// TIA Portal project "Programa" (V19)

(* hardware
DEVICE "S7-1200 station_1"  S7-1200 Station
   slot 0: "Rack_0"  S7-1200 Rack  Rack  V1.0
   slot 1: "PLC_1"  CPU 1212C DC/DC/DC  6ES7 212-1AE40-0XB0  V4.6
DEVICE "HMI_1"  KTP400 Basic PN
   slot 0: "HMI_1"  KTP400 Basic PN  6AV2 123-2DB03-0AX0  15.1.0.0
   slot 1: "HMI_RT_1"  KTP400 Basic PN  6AV2 123-2DB03-0AX0  15.1.0.0
   slot 5: "HMI_1.IE_CP_1"  PROFINET Interface  15.0.1.0
      slot 1: "Interfaz PROFINET_1"  PROFINET Interface
         slot 1: "Port_1"  Port
*)

// ===== PLC "PLC_1"  CPU 1212C DC/DC/DC =====

VAR_GLOBAL   // PLC tag table "Default tag table"
   "Pulsador_2" AT %I0.0 : Bool;
   "Luz_2_G" AT %Q0.3 : Bool;
   "Pulsador_1" AT %I0.4 : Bool;
   "Luz_1_Y" AT %Q0.4 : Bool;
   "Paro_Emergencia" AT %I0.1 : Bool;
   "Pulsador_Stop" AT %I0.3 : Bool;
   "Pulsador_Start" AT %I0.2 : Bool;
   "Potenciometro_1" AT %IW64 : Int;
   "Potenciometro_2" AT %IW66 : Int;
   "Valor_Pot_1" AT %MD56 : Real;
   "Voltaje_1" AT %MD34 : Real;
   "Valor_Pot_2" AT %MD38 : Real;
   "Voltaje_2" AT %MD46 : Real;
   "Eje_1_Impulso" AT %Q0.0 : Bool;
   "Eje_1_Sentido" AT %Q0.1 : Bool;
   "Eje_1_HabilitarAccionamiento" AT %Q0.2 : Bool;
   "System_Byte" AT %MB1 : Byte;
   "FirstScan" AT %M1.0 : Bool;
   "DiagStatusUpdate" AT %M1.1 : Bool;
   "AlwaysTRUE" AT %M1.2 : Bool;
   "AlwaysFALSE" AT %M1.3 : Bool;
   "Clock_Byte" AT %MB0 : Byte;
   "Clock_10Hz" AT %M0.0 : Bool;
   "Clock_5Hz" AT %M0.1 : Bool;
   "Clock_2.5Hz" AT %M0.2 : Bool;
   "Clock_2Hz" AT %M0.3 : Bool;
   "Clock_1.25Hz" AT %M0.4 : Bool;
   "Clock_1Hz" AT %M0.5 : Bool;
   "Clock_0.625Hz" AT %M0.6 : Bool;
   "Clock_0.5Hz" AT %M0.7 : Bool;
   "Activación_Motor" AT %M2.0 : Bool;
   "Dirección_Motor" AT %M2.1 : Bool;
   "Set_Home" AT %M2.2 : Bool;
   "Detención_Eje" AT %M2.3 : Bool;
   "Activación_Modo_Relativo" AT %M2.4 : Bool;
   "Rotación_Motor" AT %MD10 : Real;
   "Velocidad_Motor" AT %MD14 : Real;
   "Activación_Modo_Absoluto" AT %M2.5 : Bool;
   "Tag_7" AT %MD18 : Real;
   "Tag_8" AT %MD22 : Real;
   "Activacion_Modo_Velocidad" AT %M2.6 : Bool;
   "Dir_Motor" AT %MW26 : Int;
   "Dirección_Izquierda" AT %M3.0 : Bool;
   "Dirección_Derecha" AT %M3.1 : Bool;
   "HMI_Activación" AT %M3.2 : Bool;
   "Vel_Norm" AT %MW28 : Int;
   "Set_vel_Norm" AT %MW30 : Int;
   "Luz_3_R" AT %Q0.5 : Bool;
   "Luz_Verde" AT %M3.3 : Bool;
   "Luz_Amarilla" AT %M3.4 : Bool;
   "Luz_Roja" AT %M3.5 : Bool;
   "Eje_Detenido" AT %M3.6 : Bool;
   "Eje_Trabajando" AT %M3.7 : Bool;
   "Izq_HMI" AT %M4.0 : Bool;
   "Der_HMI" AT %M4.1 : Bool;
   "Pulsos_Nor" AT %MD42 : Real;
   "Rotacion_Norm" AT %MW50 : Int;
   "Activar_Pot" AT %M4.2 : Bool;
   "Vel_pot" AT %MW52 : Int;
END_VAR

DATA_BLOCK "Eje_1"   // DB1, Motion_DB
{ S7_Optimized_Access := 'TRUE' }
AUTHOR : SIMATIC
FAMILY : BasicMC
NAME : TO_PosAx
VERSION : 8.0
// stored: InstanceOfName TO_PositioningAxis
"TO_PositioningAxis"
BEGIN
   // Axis.EnableOutput_AddressCU = %Q0.2
   // Axis.LengthUnit.LastDistance = -1
   // Axis.OnlinePtoModeCU = 16#0000_0002
   // Axis.DirectionOutputEnabledCU = TRUE
   // Axis.SelectedChannel2EnumCU = %Q0.1
   // Axis.SelectedChannel1EnumCU = %Q0.0
   // Pulse.MinDeltaDeltaFrequencyCU = 0.004
   // Pulse.MaxDeltaDeltaFrequencyCU = 1.0E+10
   // Pulse.MinDeltaFrequencyCU = 0.005
   // Pulse.MaxDeltaFrequencyCU = 9.5E+9
   // Pulse.MinFrequencyCU = 1.0
   // Pulse.MaxFrequencyCU = 100000.0
   // Pulse.OutputSourceCU = 16#0000_0000
   // Axis.SelectPTO = 0
END_DATA_BLOCK

ORGANIZATION_BLOCK "Main"   // OB1, LAD, ProgramCycle
TITLE = "Main Program Sweep (Cycle)"
{ S7_Optimized_Access := 'TRUE' }
VERSION : 0.1
   VAR_INPUT
      Initial_Call : Bool;   // Initial call of this OB
      Remanence : Bool;   // =True, if remanent data are available
   END_VAR
BEGIN

REGION Network 1
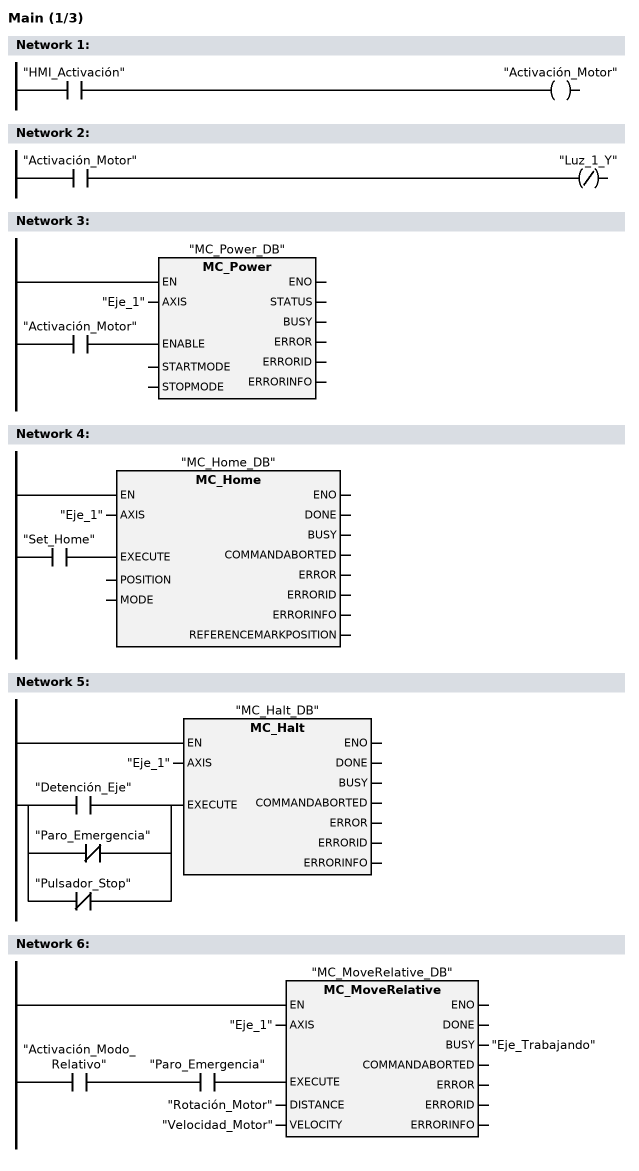
   RUNG wire#powerrail
      Contact( "HMI_Activación" )
      Coil( "Activación_Motor" )
   END_RUNG
   // the same network as SCL:
   "Activación_Motor" := "HMI_Activación";
END_REGION

REGION Network 2
   RUNG wire#powerrail
      Contact( "Activación_Motor" )
      I_Coil( "Luz_1_Y" )
   END_RUNG
   // the same network as SCL:
   "Luz_1_Y" := NOT "Activación_Motor";
END_REGION

REGION Network 3
   "MC_Power_DB"(Axis := "Eje_1", Enable := "Activación_Motor");   // MC_Power
END_REGION

REGION Network 4
   "MC_Home_DB"(Axis := "Eje_1", Execute := "Set_Home");   // MC_Home
END_REGION

REGION Network 5
   "MC_Halt_DB"(Axis := "Eje_1", Execute := "Detención_Eje" OR NOT "Paro_Emergencia" OR NOT "Pulsador_Stop");   // MC_Halt
END_REGION

REGION Network 6
   "MC_MoveRelative_DB"(Axis := "Eje_1",   // MC_MoveRelative
                        Execute := "Activación_Modo_Relativo" AND "Paro_Emergencia",
                        Distance := "Rotación_Motor",
                        Velocity := "Velocidad_Motor",
                        Busy => "Eje_Trabajando");
END_REGION

REGION Network 7
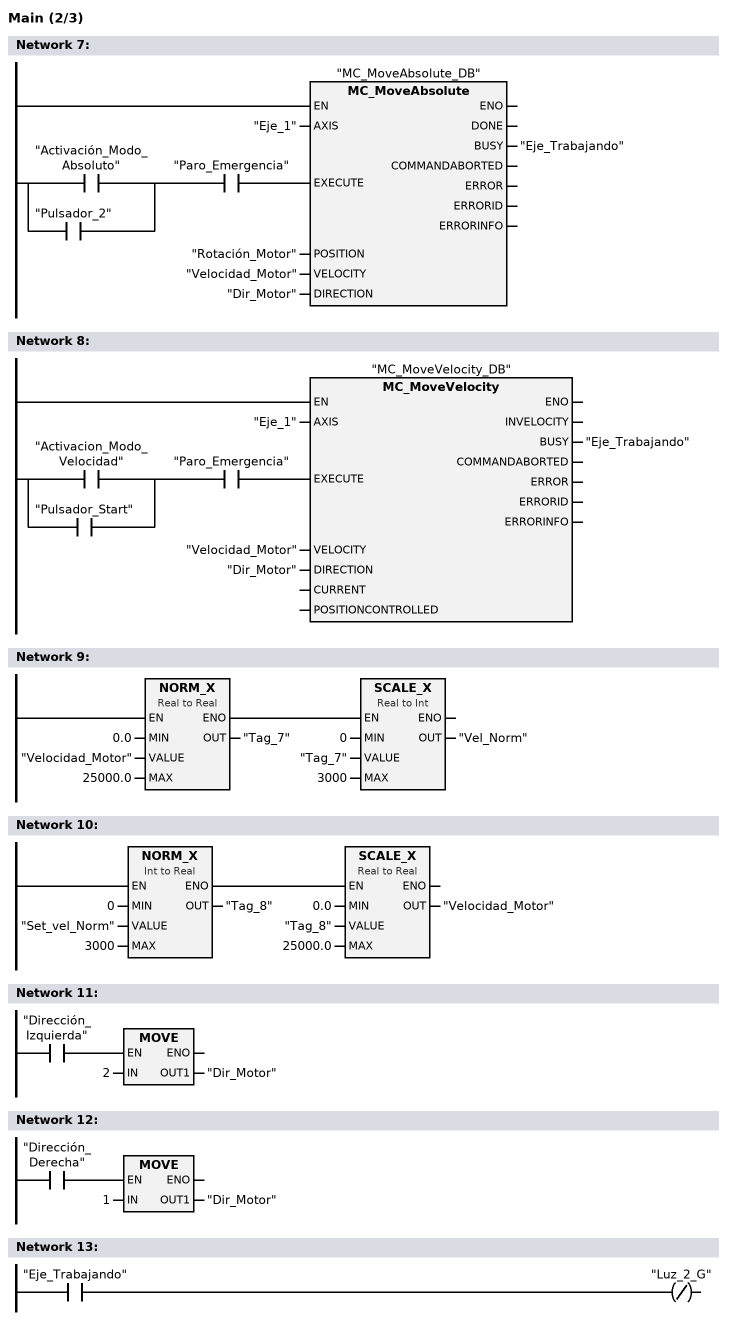
   "MC_MoveAbsolute_DB"(Axis := "Eje_1",   // MC_MoveAbsolute
                        Execute := ("Activación_Modo_Absoluto" OR "Pulsador_2") AND "Paro_Emergencia",
                        Position := "Rotación_Motor",
                        Velocity := "Velocidad_Motor",
                        Direction := "Dir_Motor",
                        Busy => "Eje_Trabajando");
END_REGION

REGION Network 8
   "MC_MoveVelocity_DB"(Axis := "Eje_1",   // MC_MoveVelocity
                        Execute := ("Activacion_Modo_Velocidad" OR "Pulsador_Start") AND "Paro_Emergencia",
                        Velocity := "Velocidad_Motor",
                        Direction := "Dir_Motor",
                        Busy => "Eje_Trabajando");
END_REGION

REGION Network 9
   RUNG wire#powerrail
      { S7_Templates := "[SrcType := Real, DestType := Real]" } Normalize(min := 0.0, value := "Velocidad_Motor", max := 25000.0, out => "Tag_7")
      { S7_Templates := "[SrcType := Real, DestType := Int]" } Scale(min := 0, value := "Tag_7", max := 3000, out => "Vel_Norm")
   END_RUNG
   // the same network as SCL:
   "Tag_7" := NORM_X(MIN := 0.0, VALUE := "Velocidad_Motor", MAX := 25000.0);
   "Vel_Norm" := SCALE_X(MIN := 0, VALUE := "Tag_7", MAX := 3000);
END_REGION

REGION Network 10
   RUNG wire#powerrail
      { S7_Templates := "[SrcType := Int, DestType := Real]" } Normalize(min := 0, value := "Set_vel_Norm", max := 3000, out => "Tag_8")
      { S7_Templates := "[SrcType := Real, DestType := Real]" } Scale(min := 0.0, value := "Tag_8", max := 25000.0, out => "Velocidad_Motor")
   END_RUNG
   // the same network as SCL:
   "Tag_8" := NORM_X(MIN := 0, VALUE := "Set_vel_Norm", MAX := 3000);
   "Velocidad_Motor" := SCALE_X(MIN := 0.0, VALUE := "Tag_8", MAX := 25000.0);
END_REGION

REGION Network 11
   RUNG wire#powerrail
      Contact( "Dirección_Izquierda" )
      Move(in := 2, out1 => "Dir_Motor")
   END_RUNG
   // the same network as SCL:
   IF "Dirección_Izquierda" THEN "Dir_Motor" := 2; END_IF;
END_REGION

REGION Network 12
   RUNG wire#powerrail
      Contact( "Dirección_Derecha" )
      Move(in := 1, out1 => "Dir_Motor")
   END_RUNG
   // the same network as SCL:
   IF "Dirección_Derecha" THEN "Dir_Motor" := 1; END_IF;
END_REGION

REGION Network 13
   RUNG wire#powerrail
      Contact( "Eje_Trabajando" )
      I_Coil( "Luz_2_G" )
   END_RUNG
   // the same network as SCL:
   "Luz_2_G" := NOT "Eje_Trabajando";
END_REGION

REGION Network 14
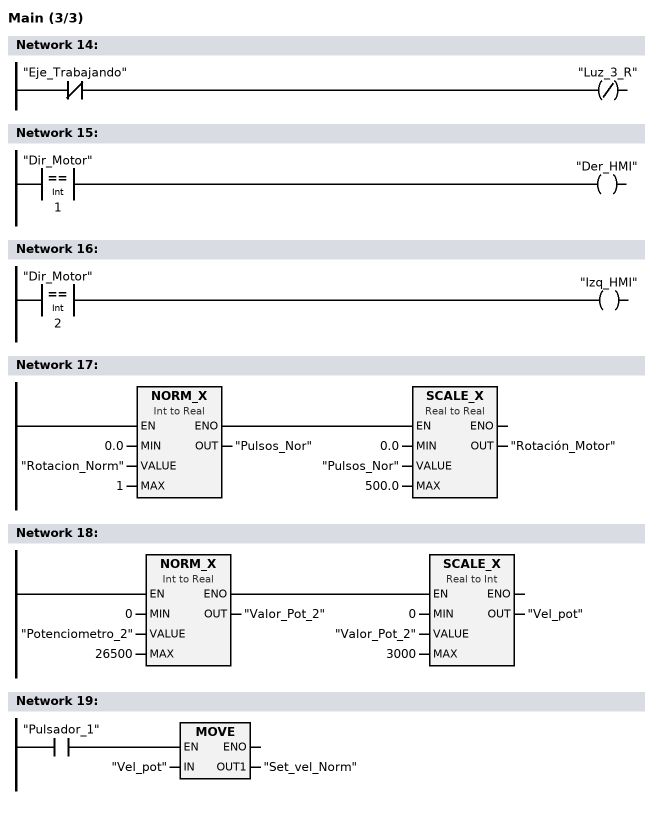
   RUNG wire#powerrail
      I_Contact( "Eje_Trabajando" )
      I_Coil( "Luz_3_R" )
   END_RUNG
   // the same network as SCL:
   "Luz_3_R" := NOT (NOT "Eje_Trabajando");
END_REGION

REGION Network 15
   RUNG wire#powerrail
      { S7_Templates := "SrcType := Int" } EQ_Contact(in1 := "Dir_Motor", in2 := 1)
      Coil( "Der_HMI" )
   END_RUNG
   // the same network as SCL:
   "Der_HMI" := "Dir_Motor" = 1;
END_REGION

REGION Network 16
   RUNG wire#powerrail
      { S7_Templates := "SrcType := Int" } EQ_Contact(in1 := "Dir_Motor", in2 := 2)
      Coil( "Izq_HMI" )
   END_RUNG
   // the same network as SCL:
   "Izq_HMI" := "Dir_Motor" = 2;
END_REGION

REGION Network 17
   RUNG wire#powerrail
      { S7_Templates := "[SrcType := Int, DestType := Real]" } Normalize(min := 0.0, value := "Rotacion_Norm", max := 1, out => "Pulsos_Nor")
      { S7_Templates := "[SrcType := Real, DestType := Real]" } Scale(min := 0.0, value := "Pulsos_Nor", max := 500.0, out => "Rotación_Motor")
   END_RUNG
   // the same network as SCL:
   "Pulsos_Nor" := NORM_X(MIN := 0.0, VALUE := "Rotacion_Norm", MAX := 1);
   "Rotación_Motor" := SCALE_X(MIN := 0.0, VALUE := "Pulsos_Nor", MAX := 500.0);
END_REGION

REGION Network 18
   RUNG wire#powerrail
      { S7_Templates := "[SrcType := Int, DestType := Real]" } Normalize(min := 0, value := "Potenciometro_2", max := 26500, out => "Valor_Pot_2")
      { S7_Templates := "[SrcType := Real, DestType := Int]" } Scale(min := 0, value := "Valor_Pot_2", max := 3000, out => "Vel_pot")
   END_RUNG
   // the same network as SCL:
   "Valor_Pot_2" := NORM_X(MIN := 0, VALUE := "Potenciometro_2", MAX := 26500);
   "Vel_pot" := SCALE_X(MIN := 0, VALUE := "Valor_Pot_2", MAX := 3000);
END_REGION

REGION Network 19
   RUNG wire#powerrail
      Contact( "Pulsador_1" )
      Move(in := "Vel_pot", out1 => "Set_vel_Norm")
   END_RUNG
   // the same network as SCL:
   IF "Pulsador_1" THEN "Set_vel_Norm" := "Vel_pot"; END_IF;
END_REGION
END_ORGANIZATION_BLOCK

(* ===== HMI "HMI_RT_1" =====
system functions are stored by id; their names below are inferred from use
connection "HMI_Conexión_1": ETHERNET, SMART_S7_1200_OMS

HMI tags "Tabla de variables estándar"
   "Activación_Motor" : Bool = PLC Activación_Motor AT %M2.0, 1 s
   "Dirección_Motor" : Bool = PLC Dirección_Motor AT %M2.1, 1 s
   "Tag_2" : Bool = PLC Detención_Eje AT %M2.3, 1 s
   "Velocidad_Motor" : Real = PLC Velocidad_Motor AT %MD14, 1 s
   "Rotación_Motor" : Real = PLC Rotación_Motor AT %MD10, 1 s
   "Tag_3" : Bool = PLC Activación_Modo_Relativo AT %M2.4, 1 s
   "Tag_9" : Bool = PLC Activacion_Modo_Velocidad AT %M2.6, 1 s
   "Dirección_Izquierda" : Bool = PLC Dirección_Derecha AT %M3.1, 1 s
   "Dirección_Derecha" : Bool = PLC Dirección_Izquierda AT %M3.0, 1 s
   "HMI_Activación" : Bool = PLC HMI_Activación AT %M3.2, 1 s
   "Dir_Motor" : Int = PLC Dir_Motor AT %MW26, 1 s
   "Set_vel_Norm" : Int = PLC Set_vel_Norm AT %MW30, 1 s
   "Vel_Norm" : Int = PLC Vel_Norm AT %MW28, 1 s
   "Rotacion_Norm" : Int = PLC Rotacion_Norm AT %MW50, 1 s

screen "Imagen raíz" 480x272, template "Plantilla_1"
   Softkey "Softkey_F1" at 0,0 size 0x0
      on KeyDown: ActivateScreen("Imagen raíz", 0)
   Softkey "Softkey_F2" at 0,0 size 0x0
      on KeyDown: ActivateScreen("Control_Motor", 0)
   TextField "Campo de texto_1" at 28,22 size 192x81; Text 'Sistema de Control de un ServoMotor'
   GraphicView "Visor de gráficos_1" at 237,28 size 217x231; Picture "Gráfico_5"
   GraphicView "Visor de gráficos_2" at 33,111 size 169x144; Picture "Gráfico_6"

screen "Control_Motor" 480x272
   Softkey "Softkey_F2" at 0,0 size 0x0
      on KeyDown: ActivateScreen("Control_Motor", 0)
   Softkey "Softkey_F1" at 0,0 size 0x0
      on KeyDown: ActivateScreen("Imagen raíz", 0)
   GraphicView "Visor de gráficos_3" at 345,158 size 114x112; Picture "Motor"
   Switch "Interruptor_1" at 41,44 size 68x26; CaptionText 'Switch'; TextOff 'OFF'; TextOn 'ON'
      on SwitchOn: SetBit("HMI_Activación")
      on SwitchOff: ResetBit("HMI_Activación")
      ProcessValue <- "Activación_Motor"
   TextField "Campo de texto_1" at 18,13 size 116x20; Text 'Activación Motor'
   GraphicView "Visor de gráficos_2" at 332,212 size 50x50; Picture "Horario"
      Visibility <- "Dirección_Izquierda"
   GraphicView "Visor de gráficos_1" at 331,212 size 50x50; Picture "Antihorario"
      Visibility <- "Dirección_Derecha"
   Switch "Interruptor_2" at 40,111 size 68x26; CaptionText 'Switch'; TextOff 'Derecha'; TextOn 'Izquierda'
      on SwitchOn: SetBit("Dirección_Izquierda"); ResetBit("Dirección_Derecha")
      on SwitchOff: SetBit("Dirección_Derecha"); ResetBit("Dirección_Izquierda")
      ProcessValue <- "Dir_Motor"
   TextField "Campo de texto_2" at 111,112 size 28x20; Text 'Der'
   TextField "Campo de texto_3" at 22,83 size 107x20; Text 'Dirección Motor'
   TextField "Campo de texto_4" at 9,112 size 25x20; Text 'Izq'
   TextField "Campo de texto_5" at 111,46 size 22x20; Text 'On'
   TextField "Campo de texto_6" at 9,46 size 24x20; Text 'Off'
   TextField "Campo de texto_7" at 175,14 size 228x20; Text 'Velocidad Motor en RPM (0 -3000)'
   IOField "Campo ES_1" at 299,41 size 72x32; FormatPattern 99999
      ProcessValue <- "Set_vel_Norm"
   TextField "Campo de texto_8" at 174,142 size 105x20; Text 'Rotación de Eje'
   IOField "Campo ES_2" at 192,167 size 72x32; FormatPattern 99999
      ProcessValue <- "Rotacion_Norm"
   Button "Botón_1" at 183,212 size 93x29; TextOff 'Iniciar Giro'
      on Press: SetBit("Tag_3")
      on Release: ResetBit("Tag_3")
   Button "Botón_2" at 183,83 size 93x29; TextOff 'Detener Eje'
      on Press: SetBit("Tag_2")
      on Release: ResetBit("Tag_2")
   Bar "Barra_1" at 299,85 size 148x28; MinimumValue 0; MaximumValue 3000
      ProcessValue <- "Vel_Norm"
   Button "Botón_3" at 183,44 size 93x29; TextOff 'Mover Eje'
      on Press: SetBit("Tag_9")
      on Release: ResetBit("Tag_9")
*)